PROGRAM PRG_TEST
(*************************************************************************************************)
(*  FILENAME:    PRG_TEST.EXP                                                                    *)
(*  PROJECT:     CALMAR PUPLC                                                                    *)
(*  COPYRIGHT:   All rights reserved (c) Wifag//Polytype, Fribourg/Switzerland (2016)            *)
(*  ENVIRONMENT: TwinCAT PLC                                                                     *)
(*  VERSION:     <version>                                                                       *)
(*************************************************************************************************)
(*  DESCRIPTION:                                                                   <description> *)
(*    Controls the test functions.                                                               *)
(*                                                                                </description> *)
(*************************************************************************************************)

VAR
	bL_FirstRun           : BOOL := TRUE;

  (*Test CONFIGURATION*)


  
  (*Motion simulation*)
  _fb_sim_el5101        : FB_EL5101_SIM;
  bL_Sim_EL5101         : BOOL;   (*enable EL5001 io simulation*) 
  
END_VAR

(* INIT First action init call*)
IF bL_FirstRun THEN
	bL_FirstRun := FALSE;
	Init();
END_IF;

(*** configure tests ****************************)
(*--> un-comment the defines in GVL_TestCfg*)
(************************************************)

(*** Library testing ***)
{IF defined (variable: GVL_TestCfg.do_LibTest)}
  LibTest();
{END_IF}

ACTION Init:

; // nothing to do
END_ACTION

ACTION LibTest:
CalmarCommons.PRG_TEST();
CalmarCompPrint.PRG_TEST();
END_ACTION

END_PROGRAM

(* stored: Version 1.1.0.1, ProductVersion 3.1.4024.11
   POU PRG_TEST: Id {aa609c94-50ed-4e2d-83a1-00bb16a3be93}, SpecialFunc None
   Action Init: Id {15466f12-fe50-464a-bc06-a462dd113028}
   Action LibTest: Id {df43acd7-7245-4dbb-a1db-5e797fac5e48} *)
